(* IEC 61131-3 sources: motion-safety-bench/plc, 16 files *)

(* ---- Enumerations.st ---- *)
TYPE E_MachineMode :
(
    MODE_OFF        := 0,
    MODE_INIT       := 1,
    MODE_HOMING     := 2,
    MODE_MANUAL_JOG := 3,
    MODE_AUTO       := 4,
    MODE_FAULT      := 5,
    MODE_RESET      := 6
);
END_TYPE

TYPE E_AxisState :
(
    AXIS_DISABLED           := 0,
    AXIS_STANDSTILL         := 1,
    AXIS_HOMING             := 2,
    AXIS_DISCRETE_MOTION    := 3,
    AXIS_CONTINUOUS_MOTION  := 4,
    AXIS_STOPPING           := 5,
    AXIS_ERRORSTOP          := 6
);
END_TYPE

TYPE E_AlarmSeverity :
(
    SEV_INFO        := 0,
    SEV_WARNING     := 1,
    SEV_FAULT       := 2,
    SEV_CRITICAL    := 3
);
END_TYPE

TYPE E_AlarmState :
(
    ALARM_INACTIVE      := 0,
    ALARM_ACTIVE        := 1,
    ALARM_ACKNOWLEDGED  := 2,
    ALARM_CLEARED       := 3
);
END_TYPE

TYPE E_CommandType :
(
    CMD_NONE                := 0,
    CMD_MODE_REQUEST        := 1,
    CMD_JOG_POSITIVE        := 2,
    CMD_JOG_NEGATIVE        := 3,
    CMD_MOVE_ABSOLUTE       := 4,
    CMD_MOVE_RELATIVE       := 5,
    CMD_STOP                := 6,
    CMD_RESET               := 7,
    CMD_HOME                := 8,
    CMD_ACK_ALARM           := 9,
    CMD_RESET_ALL_ALARMS    := 10
);
END_TYPE

TYPE E_CommandStatus :
(
    CMDSTAT_IDLE        := 0,
    CMDSTAT_PENDING     := 1,
    CMDSTAT_EXECUTING   := 2,
    CMDSTAT_DONE        := 3,
    CMDSTAT_ERROR       := 4
);
END_TYPE

TYPE E_HomingState :
(
    HOM_IDLE            := 0,
    HOM_SEEKING_SWITCH  := 1,
    HOM_BACKING_OFF     := 2,
    HOM_SEEKING_INDEX   := 3,
    HOM_SETTING_POS     := 4,
    HOM_COMPLETE        := 5,
    HOM_ERROR           := 6
);
END_TYPE

TYPE E_TraceSource :
(
    TRACE_MODE      := 0,
    TRACE_AXIS      := 1,
    TRACE_HOMING    := 2,
    TRACE_SAFETY    := 3,
    TRACE_ALARM     := 4,
    TRACE_COMMAND   := 5,
    TRACE_CONFIG    := 6,
    TRACE_TEST      := 7
);
END_TYPE

TYPE E_TestPhase :
(
    TEST_IDLE       := 0,
    TEST_SETUP      := 1,
    TEST_EXECUTE    := 2,
    TEST_SETTLE     := 3,
    TEST_VERIFY     := 4,
    TEST_TEARDOWN   := 5,
    TEST_DONE       := 6
);
END_TYPE

TYPE E_TestResult :
(
    TRES_NOT_RUN    := 0,
    TRES_RUNNING    := 1,
    TRES_PASS       := 2,
    TRES_FAIL       := 3,
    TRES_TIMEOUT    := 4
);
END_TYPE

(* ---- Structures.st ---- *)
TYPE ST_AxisConfig :
STRUCT
    fMaxVelocity : LREAL := 500.0;
    fMaxAcceleration : LREAL := 2000.0;
    fMaxDeceleration : LREAL := 2000.0;
    fJerkLimit : LREAL := 10000.0;
    fSoftLimitPositive : LREAL := 300.0;
    fSoftLimitNegative : LREAL := -10.0;
    fHomingVelocity : LREAL := 50.0;
    fHomingBackoffVelocity : LREAL := 10.0;
    bHomingDirectionPositive : BOOL := FALSE;
    fHomeOffset : LREAL := 0.0;
    fPositionErrorLimit : LREAL := 2.0;
    fJogVelocity : LREAL := 100.0;
END_STRUCT
END_TYPE

TYPE ST_AxisStatus :
STRUCT
    fActualPosition : LREAL;
    fActualVelocity : LREAL;
    fActualTorque : LREAL;
    eAxisState : E_AxisState;
    bEnabled : BOOL;
    bHomed : BOOL;
    bInMotion : BOOL;
    bError : BOOL;
    nErrorCode : UDINT;
    bPositiveLimitActive : BOOL;
    bNegativeLimitActive : BOOL;
END_STRUCT
END_TYPE

TYPE ST_SafetyConfig :
STRUCT
    tEStopDebounceTime : TIME := T#100MS;
    tRelayDiscrepancyWindow : TIME := T#500MS;
    tLimitDebounceTime : TIME := T#50MS;
    tStuckSensorTimeout : TIME := T#5S;
END_STRUCT
END_TYPE

TYPE ST_SafetyStatus :
STRUCT
    bSafeToRun : BOOL;
    bEStopActive : BOOL;
    bSafetyRelayOK : BOOL;
    bRelayDiscrepancy : BOOL;
    bAnyLimitTripped : BOOL;
    abLimitPosActive : ARRAY[1..2] OF BOOL;
    abLimitNegActive : ARRAY[1..2] OF BOOL;
    nSafetyStatusWord : UINT;
END_STRUCT
END_TYPE

TYPE ST_Alarm :
STRUCT
    nID : UINT;
    eSeverity : E_AlarmSeverity;
    eState : E_AlarmState;
    sMessage : STRING(80);
    sSource : STRING(40);
    tRaiseTime : DT;
    tAckTime : DT;
    tClearTime : DT;
    bRequiresAck : BOOL;
    bSelfClearing : BOOL;
END_STRUCT
END_TYPE

TYPE ST_HMICommand :
STRUCT
    eCommandType : E_CommandType;
    nAxisIndex : UINT;
    fValue1 : LREAL;
    fValue2 : LREAL;
    eTargetMode : E_MachineMode;
    nAlarmID : UINT;
    bExecute : BOOL;
END_STRUCT
END_TYPE

TYPE ST_MotionCommand :
STRUCT
    eType : E_CommandType;
    nAxisIndex : UINT;
    fTargetPosition : LREAL;
    fDistance : LREAL;
    fVelocity : LREAL;
    bJogPositive : BOOL;
    bJogNegative : BOOL;
    bExecute : BOOL;
    eStatus : E_CommandStatus;
END_STRUCT
END_TYPE

TYPE ST_TraceEvent :
STRUCT
    tTimestamp : DT;
    eSource : E_TraceSource;
    nEventID : UINT;
    sDescription : STRING(120);
    fValue : LREAL;
END_STRUCT
END_TYPE

TYPE ST_ModePermits :
STRUCT
    bAllowMotion : BOOL;
    bAllowJog : BOOL;
    bAllowHoming : BOOL;
    bAllowAutoStart : BOOL;
    bAllowModeChange : BOOL;
    bAllowConfigEdit : BOOL;
    bAllowAlarmReset : BOOL;
END_STRUCT
END_TYPE

TYPE ST_TimingConfig :
STRUCT
    tInitTimeout : TIME := T#10S;
    tHomingTimeout : TIME := T#60S;
    tHomingStepTimeout : TIME := T#15S;
    nHomingMaxRetries : UINT := 2;
    tCommandTimeout : TIME := T#5S;
    tTestSettleTime : TIME := T#500MS;
    tTestStepTimeout : TIME := T#30S;
END_STRUCT
END_TYPE

TYPE ST_TraceConfig :
STRUCT
    nBufferSize : UINT := 1000;
    nDisplayCount : UINT := 20;
    nPendingQueueMax : UINT := 50;
END_STRUCT
END_TYPE

TYPE ST_AlarmConfig :
STRUCT
    nMaxActiveAlarms : UINT := 32;
    nMaxAlarmHistory : UINT := 200;
END_STRUCT
END_TYPE

TYPE ST_MachineConfig :
STRUCT
    bSimulationMode : BOOL := TRUE;
    astAxisConfig : ARRAY[1..2] OF ST_AxisConfig;
    stSafetyConfig : ST_SafetyConfig;
    stTimingConfig : ST_TimingConfig;
    stTraceConfig : ST_TraceConfig;
    stAlarmConfig : ST_AlarmConfig;
    nAxisCount : UINT := 2;
END_STRUCT
END_TYPE

TYPE ST_TestResult :
STRUCT
    nTestID : UINT;
    sTestName : STRING(80);
    eResult : E_TestResult;
    sExpected : STRING(120);
    sActual : STRING(120);
    tDuration : TIME;
    tTimestamp : DT;
END_STRUCT
END_TYPE

TYPE ST_HMIData :
STRUCT
    eCurrentMode : E_MachineMode;
    stModePermits : ST_ModePermits;
    astAxisStatus : ARRAY[1..2] OF ST_AxisStatus;
    stSafetyStatus : ST_SafetyStatus;
    astActiveAlarms : ARRAY[1..32] OF ST_Alarm;
    nActiveAlarmCount : UINT;
    eHighestSeverity : E_AlarmSeverity;
    astRecentEvents : ARRAY[1..20] OF ST_TraceEvent;
    eHomingState : E_HomingState;
    bSimulationMode : BOOL;
    bHMIDataStale : BOOL;
    nCycleCount : UDINT;
END_STRUCT
END_TYPE

TYPE ST_VirtualIO :
STRUCT
    bEStop : BOOL := TRUE;
    bSafetyRelayFB : BOOL := TRUE;
    abHomeSwitch : ARRAY[1..2] OF BOOL;
    abLimitPos : ARRAY[1..2] OF BOOL := [TRUE, TRUE];
    abLimitNeg : ARRAY[1..2] OF BOOL := [TRUE, TRUE];
    bSensor1 : BOOL;
    bSensor2 : BOOL;
    bReadyLamp : BOOL;
    bFaultLamp : BOOL;
    bMotionLamp : BOOL;
    bHomedLamp : BOOL;
    bSafetyRelayCmd : BOOL;
END_STRUCT
END_TYPE

(* ---- GVL_Constants.st ---- *)
VAR_GLOBAL CONSTANT
    cMAX_AXES : UINT := 2;
    cMAX_ALARMS : UINT := 32;
    cMAX_ALARM_HISTORY : UINT := 200;
    cTRACE_BUFFER_SIZE : UINT := 1000;
    cTRACE_DISPLAY_COUNT : UINT := 20;
    cTRACE_PENDING_MAX : UINT := 50;
    cMAX_TESTS : UINT := 50;
END_VAR

(* ---- GVL_IO.st ---- *)
(*
    This is the ONLY file with AT% addresses.
    All other files use symbolic names.
*)
VAR_GLOBAL
    (* Inputs *)
    bPhysEStop           AT %IX0.0 : BOOL;
    bPhysSafetyRelayFB   AT %IX0.1 : BOOL;
    bPhysHomeSwitch1     AT %IX0.2 : BOOL;
    bPhysHomeSwitch2     AT %IX0.3 : BOOL;
    bPhysLimitPos1       AT %IX0.4 : BOOL;
    bPhysLimitNeg1       AT %IX0.5 : BOOL;
    bPhysLimitPos2       AT %IX0.6 : BOOL;
    bPhysLimitNeg2       AT %IX0.7 : BOOL;
    bPhysGuardDoorClosed AT %IX1.0 : BOOL;
    bPhysSTOHealthy      AT %IX1.1 : BOOL;
    bPhysDriveReady1     AT %IX1.2 : BOOL;
    bPhysDriveReady2     AT %IX1.3 : BOOL;
    bPhysDriveFault1     AT %IX1.4 : BOOL;
    bPhysDriveFault2     AT %IX1.5 : BOOL;
    bPhysEncoderHealthy1 AT %IX1.6 : BOOL;
    bPhysEncoderHealthy2 AT %IX1.7 : BOOL;
    bPhysEtherCATOK      AT %IX2.0 : BOOL;
    bPhysWatchdogOK      AT %IX2.1 : BOOL;

    (* Outputs *)
    bPhysReadyLamp       AT %QX0.0 : BOOL;
    bPhysFaultLamp       AT %QX0.1 : BOOL;
    bPhysMotionLamp      AT %QX0.2 : BOOL;
    bPhysHomedLamp       AT %QX0.3 : BOOL;
    bPhysSafetyRelayCmd  AT %QX0.4 : BOOL;
END_VAR

(* ---- GVL_VirtualIO.st ---- *)
VAR_GLOBAL
    (* Written by TestHarness or simulation environment. bSimulationMode must be TRUE. *)
    stVirtualIO : ST_VirtualIO;
END_VAR

(* ---- AlarmManager.st ---- *)
FUNCTION_BLOCK FB_AlarmManager
VAR_INPUT
    stSafetyStatus      : ST_SafetyStatus;
    bAnyAxisError       : BOOL;
    bHomingError        : BOOL;
    bConfigInvalid      : BOOL;
    bAckRequested       : BOOL;
    nAckAlarmID         : UINT;
    bResetAllRequested  : BOOL;
END_VAR

VAR_OUTPUT
    bAnyFaultActive     : BOOL;
    bAnyAlarmActive     : BOOL;
    nActiveAlarmCount   : UINT;
    eHighestSeverity    : E_AlarmSeverity;
    astActiveAlarms     : ARRAY[1..32] OF ST_Alarm;
END_VAR

VAR
    astAlarmBuffer      : ARRAY[1..32] OF ST_Alarm;
    astHistory          : ARRAY[1..200] OF ST_Alarm;
    nWriteIdx           : UINT;
    nHistoryIdx         : UINT;
END_VAR

(* ========== CONDITION EVALUATION ========== *)
METHOD EvaluateConditions
(* Method: EvaluateConditions — Purpose: Check all alarm source conditions, raise alarms as needed *)
(* TODO: IF NOT stSafetyStatus.bSafeToRun AND stSafetyStatus.bEStopActive THEN RaiseAlarm(1001, SEV_CRITICAL, 'E-stop active', 'SafetyManager', TRUE) *)
(* TODO: IF stSafetyStatus.bRelayDiscrepancy THEN RaiseAlarm(1002, SEV_CRITICAL, 'Safety relay discrepancy', 'SafetyManager', TRUE) *)
(* TODO: IF stSafetyStatus.bAnyLimitTripped THEN RaiseAlarm(1003, SEV_FAULT, 'Limit switch tripped', 'SafetyManager', TRUE) *)
(* TODO: IF bAnyAxisError THEN RaiseAlarm(2001, SEV_FAULT, 'Axis error', 'AxisManager', TRUE) *)
(* TODO: IF bHomingError THEN RaiseAlarm(3001, SEV_FAULT, 'Homing failed', 'HomingManager', TRUE) *)
END_METHOD

(* ========== OUTPUTS ========== *)
METHOD UpdateOutputs
(* Method: UpdateOutputs — Purpose: Update bAnyFaultActive, counts, highest severity *)
(* TODO: iterate astAlarmBuffer, count ACTIVE alarms, find highest severity *)
(* TODO: set bAnyFaultActive := any alarm with eSeverity >= SEV_FAULT is ACTIVE and unacknowledged *)
(* TODO: copy active alarms to astActiveAlarms output *)
END_METHOD

(* ========== RAISE ALARM ========== *)
METHOD RaiseAlarm
VAR_INPUT
    nID         : UINT;
    eSeverity   : E_AlarmSeverity;
    sMessage    : STRING(80);
    sSource     : STRING(40);
    bRequiresAck: BOOL;
END_VAR
(* Method: RaiseAlarm — Purpose: Add or update alarm in buffer with timestamp *)
(* TODO: check if alarm nID already active, if not find empty slot and populate *)
(* TODO: set tRaiseTime := NOW_DT(), eState := ALARM_ACTIVE *)
END_METHOD

(* ========== ACKNOWLEDGE ALARM ========== *)
METHOD AcknowledgeAlarm
VAR_INPUT
    nAlarmID : UINT;
END_VAR
(* Method: AcknowledgeAlarm — Purpose: Transition alarm from ACTIVE to ACKNOWLEDGED *)
(* TODO: find alarm by nID, if eState=ALARM_ACTIVE set eState:=ALARM_ACKNOWLEDGED, tAckTime:=NOW_DT() *)
END_METHOD

(* ========== RESET ALARM ========== *)
METHOD ResetAlarm
VAR_INPUT
    nAlarmID : UINT;
END_VAR
(* Method: ResetAlarm — Purpose: Clear alarm if condition is gone *)
(* TODO: find alarm by nID, if NOT bRequiresAck or already ACKNOWLEDGED, set eState:=ALARM_CLEARED *)
END_METHOD

(* ========== RESET ALL ALARMS ========== *)
METHOD ResetAllAlarms
(* Method: ResetAllAlarms — Purpose: Clear all clearable alarms *)
(* TODO: iterate buffer, call ResetAlarm on each *)
END_METHOD

END_FUNCTION_BLOCK

(* ---- CommandParser.st ---- *)
FUNCTION_BLOCK FB_CommandParser
VAR_INPUT
    stHMICommand    : ST_HMICommand;
    eCurrentMode    : E_MachineMode;
    stModePermits   : ST_ModePermits;
    stSafetyStatus  : ST_SafetyStatus;
END_VAR

VAR_OUTPUT
    eRequestedMode      : E_MachineMode;
    stMotionCommand     : ST_MotionCommand;
    bStartHoming        : BOOL;
    bAbortHoming        : BOOL;
    bAckRequested       : BOOL;
    nAckAlarmID         : UINT;
    bResetRequested     : BOOL;
    bResetAllRequested  : BOOL;
    eLastCommandStatus  : E_CommandStatus;
    sLastCommandError   : STRING(120);
END_VAR

VAR
    eProcessingState    : E_CommandStatus;
    rtrigExecute        : R_TRIG;
    nCommandCounter     : UDINT;
    nRejectedCounter    : UDINT;
END_VAR

METHOD Cyclic
(* Method: Cyclic - Purpose: Detect rising edge on bExecute, validate, route command *)

rtrigExecute(CLK := stHMICommand.bExecute);

IF rtrigExecute.Q THEN
    nCommandCounter := nCommandCounter + 1;
    IF ValidateCommand() THEN
        eLastCommandStatus := CMDSTAT_EXECUTING;
        sLastCommandError := '';

        CASE stHMICommand.eCommandType OF
            CMD_MODE_REQUEST:
                eRequestedMode := stHMICommand.eTargetMode;

            CMD_JOG_POSITIVE, CMD_JOG_NEGATIVE, CMD_MOVE_ABSOLUTE, CMD_MOVE_RELATIVE, CMD_STOP:
                stMotionCommand.eType := stHMICommand.eCommandType;
                stMotionCommand.nAxisIndex := stHMICommand.nAxisIndex;
                stMotionCommand.fTargetPosition := stHMICommand.fValue1;
                stMotionCommand.fDistance := stHMICommand.fValue1;
                stMotionCommand.fVelocity := stHMICommand.fValue2;
                stMotionCommand.bExecute := TRUE;

            CMD_HOME:
                bStartHoming := TRUE;

            CMD_RESET:
                bResetRequested := TRUE;

            CMD_ACK_ALARM:
                bAckRequested := TRUE;
                nAckAlarmID := stHMICommand.nAlarmID;

            CMD_RESET_ALL_ALARMS:
                bResetAllRequested := TRUE;
        END_CASE
    ELSE
        eLastCommandStatus := CMDSTAT_ERROR;
        nRejectedCounter := nRejectedCounter + 1;
    END_IF
ELSE
    (* Reset single-cycle triggers *)
    bStartHoming := FALSE;
    bResetRequested := FALSE;
    bAckRequested := FALSE;
    bResetAllRequested := FALSE;
    IF stMotionCommand.eType <> CMD_JOG_POSITIVE AND stMotionCommand.eType <> CMD_JOG_NEGATIVE THEN
        stMotionCommand.bExecute := FALSE;
    ELSE
        (* Keep jog active if bExecute is still true in the input struct *)
        stMotionCommand.bExecute := stHMICommand.bExecute;
    END_IF
END_IF

END_METHOD

METHOD ValidateCommand : BOOL
(* Method: ValidateCommand - Purpose: Check if command allowed in current mode and safety state *)

ValidateCommand := FALSE;

CASE stHMICommand.eCommandType OF
    CMD_MODE_REQUEST:
        IF stModePermits.bAllowModeChange THEN
            ValidateCommand := TRUE;
        ELSE
            sLastCommandError := 'Mode change not permitted';
        END_IF

    CMD_JOG_POSITIVE, CMD_JOG_NEGATIVE:
        IF stModePermits.bAllowJog AND stSafetyStatus.bSafeToRun THEN
            ValidateCommand := TRUE;
        ELSE
            sLastCommandError := 'Jog not permitted or safety not OK';
        END_IF

    CMD_MOVE_ABSOLUTE, CMD_MOVE_RELATIVE:
        IF stModePermits.bAllowMotion AND stSafetyStatus.bSafeToRun THEN
            ValidateCommand := TRUE;
        ELSE
            sLastCommandError := 'Motion not permitted or safety not OK';
        END_IF

    CMD_STOP:
        ValidateCommand := TRUE;

    CMD_HOME:
        IF stModePermits.bAllowHoming THEN
            ValidateCommand := TRUE;
        ELSE
            sLastCommandError := 'Homing not permitted';
        END_IF

    CMD_RESET, CMD_ACK_ALARM, CMD_RESET_ALL_ALARMS:
        IF stModePermits.bAllowAlarmReset THEN
            ValidateCommand := TRUE;
        ELSE
             sLastCommandError := 'Reset not permitted';
        END_IF

    CMD_NONE:
        ValidateCommand := TRUE;
END_CASE

END_METHOD

END_FUNCTION_BLOCK

(* ---- ConfigPackage.st ---- *)
FUNCTION_BLOCK FB_ConfigPackage
VAR_OUTPUT
    stMachineConfig : ST_MachineConfig;
    bSimulationMode : BOOL;
    bConfigValid    : BOOL;
    bConfigChanged  : BOOL;
END_VAR

VAR
    bInitialized    : BOOL;
    stPrevConfig    : ST_MachineConfig;
END_VAR

(* ========== CYCLIC PROCESSING ========== *)
METHOD Cyclic
(* Method: Cyclic — Purpose: Detect config changes, validate on change, set bConfigValid *)
(* TODO: compare stMachineConfig to stPrevConfig, if different set bConfigChanged, call ValidateAll *)
(* TODO: set bSimulationMode := stMachineConfig.bSimulationMode *)
END_METHOD

(* ========== DEFAULT CONFIGURATION ========== *)
METHOD LoadDefaults
(* Method: LoadDefaults — Purpose: Set all stMachineConfig fields to SDS default values *)
(* TODO: set stMachineConfig.bSimulationMode := TRUE *)
(* TODO: set stMachineConfig.nAxisCount := 2 *)
(* TODO: set axis config defaults per ST_AxisConfig field defaults from SDS *)
(* TODO: set stMachineConfig.stSafetyConfig to ST_SafetyConfig defaults *)
(* TODO: set stMachineConfig.stTimingConfig to ST_TimingConfig defaults *)
(* TODO: set bInitialized := TRUE *)
END_METHOD

(* ========== VALIDATION ========== *)
METHOD ValidateAll : BOOL
(* Method: ValidateAll — Purpose: Check all parameters, clamp or flag invalid values *)
(* Returns TRUE if all valid *)
(* TODO: check fMaxVelocity > 0 for each axis *)
(* TODO: check fSoftLimitPositive > fSoftLimitNegative for each axis *)
(* TODO: check all TIME values > T#0S *)
(* TODO: set bConfigValid := result *)
END_METHOD

(* ========== ACCESSORS ========== *)
METHOD GetAxisConfig : ST_AxisConfig
VAR_INPUT
    nAxisIndex : UINT;
END_VAR
(* Method: GetAxisConfig — Purpose: Return config for specific axis index *)
(* TODO: bounds check nAxisIndex against cMAX_AXES, return stMachineConfig.astAxisConfig[nAxisIndex] *)
END_METHOD

END_FUNCTION_BLOCK

(* ---- HMIModel.st ---- *)
FUNCTION_BLOCK FB_HMIModel
VAR_INPUT
    eCurrentMode : E_MachineMode;
    stModePermits : ST_ModePermits;
    astAxisStatus : ARRAY[1..2] OF ST_AxisStatus;
    stSafetyStatus : ST_SafetyStatus;
    astActiveAlarms : ARRAY[1..32] OF ST_Alarm;
    nActiveAlarmCount : UINT;
    eHighestSeverity : E_AlarmSeverity;
    astRecentEvents : ARRAY[1..20] OF ST_TraceEvent;
    eHomingState : E_HomingState;
    bSimulationMode : BOOL;
    bPLCHeartbeat : BOOL;
END_VAR
VAR_OUTPUT
    stHMIData : ST_HMIData;
    stHMICommand : ST_HMICommand;
END_VAR
VAR
    tonDataStale : TON;
    bPreviousHeartbeat : BOOL;
    bHeartbeatChanged : BOOL;
END_VAR

bHeartbeatChanged := bPLCHeartbeat <> bPreviousHeartbeat;
IF bHeartbeatChanged THEN
    bPreviousHeartbeat := bPLCHeartbeat;
END_IF
tonDataStale(IN := NOT bHeartbeatChanged, PT := T#2S);

stHMIData.eCurrentMode := eCurrentMode;
stHMIData.stModePermits := stModePermits;
stHMIData.astAxisStatus := astAxisStatus;
stHMIData.stSafetyStatus := stSafetyStatus;
stHMIData.astActiveAlarms := astActiveAlarms;
stHMIData.nActiveAlarmCount := nActiveAlarmCount;
stHMIData.eHighestSeverity := eHighestSeverity;
stHMIData.astRecentEvents := astRecentEvents;
stHMIData.eHomingState := eHomingState;
stHMIData.bSimulationMode := bSimulationMode;
stHMIData.bHMIDataStale := tonDataStale.Q;
stHMIData.nCycleCount := stHMIData.nCycleCount + 1;

END_FUNCTION_BLOCK

(* ---- ModeManager.st ---- *)
FUNCTION_BLOCK FB_ModeManager
VAR_INPUT
    stSafetyStatus      : ST_SafetyStatus;
    bAnyFaultActive     : BOOL;
    bAllAxesReady       : BOOL;
    bAllAxesHomed       : BOOL;
    eRequestedMode      : E_MachineMode;
    bResetRequested     : BOOL;
END_VAR

VAR_OUTPUT
    eCurrentMode            : E_MachineMode;
    ePreviousMode           : E_MachineMode;
    bModeTransitionActive   : BOOL;
    stModePermits           : ST_ModePermits;
END_VAR

VAR
    eInternalMode       : E_MachineMode;
    tonInitTimeout      : TON;
    tonHomingTimeout    : TON;
    bTransitionValid    : BOOL;
    rtrigModeRequest    : R_TRIG;
    rtrigResetRequest   : R_TRIG;
END_VAR

(* ========== CYCLIC PROCESSING ========== *)
METHOD Cyclic
(* Method: Cyclic — Purpose: Evaluate state machine, apply safety override, update permits *)

(* ========== SAFETY OVERRIDE (runs before CASE) ========== *)
(* TODO: IF NOT stSafetyStatus.bSafeToRun AND eInternalMode <> MODE_OFF AND eInternalMode <> MODE_FAULT THEN *)
(*           ePreviousMode := eInternalMode; eInternalMode := MODE_FAULT; END_IF *)

(* ========== STATE MACHINE ========== *)
CASE eInternalMode OF
    MODE_OFF:
        (* TODO: if StartCommand received and power healthy, transition to MODE_INIT *)
    MODE_INIT:
        (* TODO: run init timeout timer *)
        (* TODO: if init complete (axes ready, config valid, safety OK, no faults): stay in INIT awaiting homing request *)
        (* TODO: if HomingRequest and no faults: transition to MODE_HOMING *)
        (* TODO: if timeout: transition to MODE_FAULT *)
    MODE_HOMING:
        (* TODO: run homing timeout timer *)
        (* TODO: if bAllAxesHomed: transition to MODE_MANUAL_JOG *)
        (* TODO: if timeout or fault: transition to MODE_FAULT *)
    MODE_MANUAL_JOG:
        (* TODO: if AutoRequest and bAllAxesHomed: transition to MODE_AUTO *)
        (* TODO: if ReHomeRequest: transition to MODE_HOMING *)
        (* TODO: if bAnyFaultActive: transition to MODE_FAULT *)
    MODE_AUTO:
        (* TODO: if ManualRequest: transition to MODE_MANUAL_JOG (after axis stops) *)
        (* TODO: if bAnyFaultActive: transition to MODE_FAULT *)
    MODE_FAULT:
        (* TODO: latch — only exit via RESET when operator acknowledges *)
    MODE_RESET:
        (* TODO: 2s settle, re-check, transition to MODE_INIT or back to MODE_FAULT *)
END_CASE

(* TODO: eCurrentMode := eInternalMode *)
(* TODO: call UpdatePermits *)
END_METHOD

(* ========== TRANSITION VALIDATION ========== *)
METHOD ValidateTransition : BOOL
VAR_INPUT
    eFrom : E_MachineMode;
    eTo   : E_MachineMode;
END_VAR
(* Method: ValidateTransition — Purpose: Return TRUE if transition is valid per state table *)
(* TODO: CASE eFrom with nested IF on eTo checking all valid transitions from SDS Section 4.1 *)
END_METHOD

(* ========== MODE PERMITS ========== *)
METHOD UpdatePermits
(* Method: UpdatePermits — Purpose: Set stModePermits fields based on eCurrentMode *)
(* TODO: CASE eCurrentMode:
    MODE_MANUAL_JOG: bAllowMotion:=TRUE, bAllowJog:=TRUE, bAllowHoming:=TRUE, bAllowAutoStart:=TRUE
    MODE_AUTO: bAllowMotion:=TRUE, bAllowAutoStart:=FALSE (running), bAllowJog:=FALSE
    MODE_OFF: bAllowConfigEdit:=TRUE, rest FALSE
    all others: all FALSE except bAllowAlarmReset in FAULT *)
END_METHOD

END_FUNCTION_BLOCK

(* ---- SafetyManager.st ---- *)
FUNCTION_BLOCK FB_SafetyManager
VAR_INPUT
    bSimulationMode     : BOOL;
    stConfig            : ST_SafetyConfig;
    abDriveReady        : ARRAY[1..2] OF BOOL;
END_VAR

VAR_OUTPUT
    stSafetyStatus      : ST_SafetyStatus;
    bSafeToRun          : BOOL;
    bEStopActive        : BOOL;
    bAnyLimitTripped    : BOOL;
END_VAR

VAR
    bEStopRaw           : BOOL;
    bRelayFBRaw         : BOOL;
    abLimitPosRaw       : ARRAY[1..2] OF BOOL;
    abLimitNegRaw       : ARRAY[1..2] OF BOOL;
    tonEStopDebounce    : TON;
    tonRelayDiscrep     : TON;
    bRelayDiscrepancy   : BOOL;
END_VAR

(* ========== CYCLIC PROCESSING ========== *)
METHOD Cyclic
(* Method: Cyclic — Purpose: Read inputs, apply debounce, compute bSafeToRun *)
(* Step 1: call ReadInputs to populate raw signals *)
(* Step 2: apply debounce timers *)
(* Step 3: check relay discrepancy *)
(* TODO: bSafeToRun := bEStopRaw AND bRelayFBRaw AND NOT bRelayDiscrepancy AND NOT bAnyLimitTripped *)
(* TODO: populate stSafetyStatus fields *)
(* TODO: set nSafetyStatusWord as bitfield of key signals *)
END_METHOD

(* ========== INPUT SELECTION ========== *)
METHOD ReadInputs
(* Method: ReadInputs — Purpose: Select virtual or physical I/O based on bSimulationMode *)
(* TODO: IF bSimulationMode THEN read from GVL_VirtualIO.stVirtualIO ELSE read from GVL_IO *)
(* Note: E-stop and limits are NC logic — TRUE = healthy, FALSE = activated *)
END_METHOD

END_FUNCTION_BLOCK

(* ---- TestHarness.st ---- *)
FUNCTION_BLOCK FB_TestHarness
VAR_INPUT
    bRunTest : BOOL;
    nTestID : UINT;
    bRunAllTests : BOOL;
    eCurrentMode : E_MachineMode;
    astAxisStatus : ARRAY[1..2] OF ST_AxisStatus;
    stSafetyStatus : ST_SafetyStatus;
    nActiveAlarmCount : UINT;
    nTraceEventCount : UDINT;
    bSimulationMode : BOOL;
END_VAR
VAR_OUTPUT
    stHMICommand : ST_HMICommand;
    stTestResult : ST_TestResult;
    astTestSummary : ARRAY[1..50] OF ST_TestResult;
    nTestsRun : UINT;
    nTestsPassed : UINT;
    nTestsFailed : UINT;
    nCurrentTestID : UINT;
    bTestSuiteRunning : BOOL;
    bTestSuiteComplete : BOOL;
END_VAR
VAR
    eTestPhase : E_TestPhase;
    nTestStep : UINT;
    nCyclesInPhase : UDINT;
    rtrigRunTest : R_TRIG;
    rtrigRunAll : R_TRIG;
    bRunSuite : BOOL;
    bVerificationPassed : BOOL;
    bFaultObserved : BOOL;
    fInitialPosition : LREAL;
    fExpectedPosition : LREAL;
    fPeakPosition : LREAL;
    fLowPosition : LREAL;
    sTestName : STRING(80);
    sExpected : STRING(120);
    sActual : STRING(120);
END_VAR

rtrigRunTest(CLK := bRunTest);
rtrigRunAll(CLK := bRunAllTests);

(* All command edges are one scan wide unless explicitly held for jog. *)
stHMICommand.bExecute := FALSE;

IF NOT bSimulationMode THEN
    bTestSuiteRunning := FALSE;
    eTestPhase := TEST_IDLE;
ELSE
    IF rtrigRunAll.Q THEN
        nTestsRun := 0;
        nTestsPassed := 0;
        nTestsFailed := 0;
        nCurrentTestID := 1;
        bRunSuite := TRUE;
        bTestSuiteRunning := TRUE;
        bTestSuiteComplete := FALSE;
        eTestPhase := TEST_SETUP;
        nTestStep := 0;
        nCyclesInPhase := 0;
    ELSIF rtrigRunTest.Q AND (nTestID >= 1) AND (nTestID <= 16) THEN
        nCurrentTestID := nTestID;
        bRunSuite := FALSE;
        bTestSuiteRunning := TRUE;
        bTestSuiteComplete := FALSE;
        eTestPhase := TEST_SETUP;
        nTestStep := 0;
        nCyclesInPhase := 0;
    END_IF

    IF bTestSuiteRunning THEN
        nCyclesInPhase := nCyclesInPhase + 1;

        CASE eTestPhase OF
            TEST_SETUP:
                GVL_VirtualIO.stVirtualIO.bEStop := TRUE;
                GVL_VirtualIO.stVirtualIO.bSafetyRelayFB := TRUE;
                GVL_VirtualIO.stVirtualIO.bGuardDoorClosed := TRUE;
                GVL_VirtualIO.stVirtualIO.bSTOHealthy := TRUE;
                GVL_VirtualIO.stVirtualIO.bEtherCATOK := TRUE;
                GVL_VirtualIO.stVirtualIO.bWatchdogOK := TRUE;
                GVL_VirtualIO.stVirtualIO.abLimitPos[1] := TRUE;
                GVL_VirtualIO.stVirtualIO.abLimitNeg[1] := TRUE;
                GVL_VirtualIO.stVirtualIO.abLimitPos[2] := TRUE;
                GVL_VirtualIO.stVirtualIO.abLimitNeg[2] := TRUE;
                GVL_VirtualIO.stVirtualIO.abDriveReady[1] := TRUE;
                GVL_VirtualIO.stVirtualIO.abDriveReady[2] := TRUE;
                GVL_VirtualIO.stVirtualIO.abDriveFault[1] := FALSE;
                GVL_VirtualIO.stVirtualIO.abDriveFault[2] := FALSE;
                GVL_VirtualIO.stVirtualIO.abEncoderHealthy[1] := TRUE;
                GVL_VirtualIO.stVirtualIO.abEncoderHealthy[2] := TRUE;
                GVL_VirtualIO.stVirtualIO.abFollowingError[1] := FALSE;
                GVL_VirtualIO.stVirtualIO.abFollowingError[2] := FALSE;
                GVL_VirtualIO.stVirtualIO.abHomeSwitch[1] := FALSE;
                GVL_VirtualIO.stVirtualIO.abHomeSwitch[2] := FALSE;

                fInitialPosition := astAxisStatus[1].fActualPosition;
                fExpectedPosition := fInitialPosition;
                fPeakPosition := fInitialPosition;
                fLowPosition := fInitialPosition;
                bVerificationPassed := FALSE;
                bFaultObserved := FALSE;

                CASE nCurrentTestID OF
                    1:
                        sTestName := 'TR01 Startup and Homing';
                        sExpected := 'Safe startup reaches MANUAL with both axes homed';
                    2:
                        sTestName := 'TR02 Absolute Move';
                        sExpected := 'Axis 1 reaches 100.0 mm';
                    3:
                        sTestName := 'TR03 Relative Move';
                        sExpected := 'Axis 1 advances by 50.0 mm';
                        fExpectedPosition := fInitialPosition + 50.0;
                    4:
                        sTestName := 'TR04 Jog Positive and Negative';
                        sExpected := 'Axis jogs both directions and stops on release';
                    5:
                        sTestName := 'TR05 Positive Limit Switch';
                        sExpected := 'Positive limit stops motion, enters FAULT, recovers';
                    6:
                        sTestName := 'TR06 Negative Limit Switch';
                        sExpected := 'Negative limit stops motion, enters FAULT, recovers';
                    7:
                        sTestName := 'TR07 E-stop During Motion';
                        sExpected := 'E-stop stops motion, enters FAULT, recovers';
                    8:
                        sTestName := 'TR08 Guard Door During Motion';
                        sExpected := 'Guard door inhibits motion, enters FAULT, recovers';
                    9:
                        sTestName := 'TR09 Drive Fault';
                        sExpected := 'Drive fault latches axis error and recovers through RESET';
                    10:
                        sTestName := 'TR10 Following Error';
                        sExpected := 'Following error is detected and recovered';
                    11:
                        sTestName := 'TR11 Encoder Feedback Loss';
                        sExpected := 'Feedback loss is detected and recovered';
                    12:
                        sTestName := 'TR12 EtherCAT Dropout';
                        sExpected := 'Network dropout inhibits motion and recovers';
                    13:
                        sTestName := 'TR13 Warm Restart';
                        sExpected := 'Stop/restart leaves no stale motion command';
                    14:
                        sTestName := 'TR14 Cold Restart Defaults';
                        sExpected := 'Virtual safe defaults are restored';
                    15:
                        sTestName := 'TR15 Watchdog Timeout';
                        sExpected := 'Watchdog loss enters FAULT and recovers';
                    16:
                        sTestName := 'TR16 Invalid Command Transition';
                        sExpected := 'Move command in OFF is rejected without motion';
                END_CASE

                stTestResult.nTestID := nCurrentTestID;
                stTestResult.sTestName := sTestName;
                stTestResult.sExpected := sExpected;
                stTestResult.eResult := TRES_RUNNING;
                eTestPhase := TEST_EXECUTE;
                nTestStep := 0;
                nCyclesInPhase := 0;

            TEST_EXECUTE:
                IF astAxisStatus[1].fActualPosition > fPeakPosition THEN
                    fPeakPosition := astAxisStatus[1].fActualPosition;
                END_IF
                IF astAxisStatus[1].fActualPosition < fLowPosition THEN
                    fLowPosition := astAxisStatus[1].fActualPosition;
                END_IF

                CASE nCurrentTestID OF
                    1:
                        IF nTestStep = 0 THEN
                            stHMICommand.eCommandType := CMD_MODE_REQUEST;
                            stHMICommand.eTargetMode := MODE_INIT;
                            stHMICommand.bExecute := TRUE;
                            nTestStep := 1;
                        ELSIF nTestStep = 1 THEN
                            nTestStep := 2;
                        ELSIF nTestStep = 2 THEN
                            stHMICommand.eCommandType := CMD_MODE_REQUEST;
                            stHMICommand.eTargetMode := MODE_HOMING;
                            stHMICommand.bExecute := TRUE;
                            nTestStep := 3;
                        ELSIF nTestStep = 3 THEN
                            nTestStep := 4;
                        ELSIF nTestStep = 4 THEN
                            stHMICommand.eCommandType := CMD_HOME;
                            stHMICommand.bExecute := TRUE;
                            nTestStep := 5;
                        ELSIF nCyclesInPhase = 20 THEN
                            GVL_VirtualIO.stVirtualIO.abHomeSwitch[1] := TRUE;
                        ELSIF nCyclesInPhase = 30 THEN
                            GVL_VirtualIO.stVirtualIO.abHomeSwitch[1] := FALSE;
                        ELSIF nCyclesInPhase = 40 THEN
                            GVL_VirtualIO.stVirtualIO.abHomeSwitch[1] := TRUE;
                        ELSIF nCyclesInPhase = 50 THEN
                            GVL_VirtualIO.stVirtualIO.abHomeSwitch[1] := FALSE;
                        ELSIF nCyclesInPhase = 60 THEN
                            GVL_VirtualIO.stVirtualIO.abHomeSwitch[2] := TRUE;
                        ELSIF nCyclesInPhase = 70 THEN
                            GVL_VirtualIO.stVirtualIO.abHomeSwitch[2] := FALSE;
                        ELSIF nCyclesInPhase = 80 THEN
                            GVL_VirtualIO.stVirtualIO.abHomeSwitch[2] := TRUE;
                        ELSIF nCyclesInPhase >= 120 THEN
                            eTestPhase := TEST_VERIFY;
                        END_IF

                    2:
                        IF nTestStep = 0 THEN
                            stHMICommand.eCommandType := CMD_MOVE_ABSOLUTE;
                            stHMICommand.nAxisIndex := 1;
                            stHMICommand.fValue1 := 100.0;
                            stHMICommand.fValue2 := 200.0;
                            stHMICommand.bExecute := TRUE;
                            nTestStep := 1;
                        ELSIF (NOT astAxisStatus[1].bInMotion) AND (nCyclesInPhase > 5) THEN
                            eTestPhase := TEST_VERIFY;
                        END_IF

                    3:
                        IF nTestStep = 0 THEN
                            stHMICommand.eCommandType := CMD_MOVE_RELATIVE;
                            stHMICommand.nAxisIndex := 1;
                            stHMICommand.fValue1 := 50.0;
                            stHMICommand.fValue2 := 200.0;
                            stHMICommand.bExecute := TRUE;
                            nTestStep := 1;
                        ELSIF (NOT astAxisStatus[1].bInMotion) AND (nCyclesInPhase > 5) THEN
                            eTestPhase := TEST_VERIFY;
                        END_IF

                    4:
                        stHMICommand.nAxisIndex := 1;
                        stHMICommand.fValue1 := 50.0;
                        IF nCyclesInPhase <= 50 THEN
                            stHMICommand.eCommandType := CMD_JOG_POSITIVE;
                            stHMICommand.bExecute := TRUE;
                        ELSIF (nCyclesInPhase >= 70) AND (nCyclesInPhase <= 120) THEN
                            stHMICommand.eCommandType := CMD_JOG_NEGATIVE;
                            stHMICommand.bExecute := TRUE;
                        ELSIF nCyclesInPhase >= 140 THEN
                            eTestPhase := TEST_VERIFY;
                        END_IF

                    5:
                        IF nTestStep = 0 THEN
                            stHMICommand.eCommandType := CMD_MOVE_ABSOLUTE;
                            stHMICommand.nAxisIndex := 1;
                            stHMICommand.fValue1 := 250.0;
                            stHMICommand.fValue2 := 100.0;
                            stHMICommand.bExecute := TRUE;
                            nTestStep := 1;
                        ELSIF (nTestStep = 1) AND (nCyclesInPhase >= 20) THEN
                            GVL_VirtualIO.stVirtualIO.abLimitPos[1] := FALSE;
                            IF (eCurrentMode = MODE_FAULT) AND (NOT astAxisStatus[1].bInMotion) THEN
                                bFaultObserved := TRUE;
                                GVL_VirtualIO.stVirtualIO.abLimitPos[1] := TRUE;
                                nTestStep := 2;
                            END_IF
                        ELSIF nTestStep = 2 THEN
                            stHMICommand.eCommandType := CMD_RESET;
                            stHMICommand.bExecute := TRUE;
                            nTestStep := 3;
                        ELSIF nTestStep = 3 THEN
                            nTestStep := 4;
                        ELSIF (nTestStep = 4) AND (nCyclesInPhase >= 90) THEN
                            stHMICommand.eCommandType := CMD_RESET_ALL_ALARMS;
                            stHMICommand.bExecute := TRUE;
                            nTestStep := 5;
                        ELSIF nTestStep = 5 THEN
                            nTestStep := 6;
                        ELSIF (nTestStep = 6) AND (nCyclesInPhase >= 140) THEN
                            stHMICommand.eCommandType := CMD_MODE_REQUEST;
                            stHMICommand.eTargetMode := MODE_MANUAL_JOG;
                            stHMICommand.bExecute := TRUE;
                            nTestStep := 7;
                        ELSIF (nTestStep = 7) AND (eCurrentMode = MODE_MANUAL_JOG) THEN
                            eTestPhase := TEST_VERIFY;
                        END_IF

                    6:
                        IF nTestStep = 0 THEN
                            stHMICommand.eCommandType := CMD_MOVE_ABSOLUTE;
                            stHMICommand.nAxisIndex := 1;
                            stHMICommand.fValue1 := -5.0;
                            stHMICommand.fValue2 := 100.0;
                            stHMICommand.bExecute := TRUE;
                            nTestStep := 1;
                        ELSIF (nTestStep = 1) AND (nCyclesInPhase >= 20) THEN
                            GVL_VirtualIO.stVirtualIO.abLimitNeg[1] := FALSE;
                            IF (eCurrentMode = MODE_FAULT) AND (NOT astAxisStatus[1].bInMotion) THEN
                                bFaultObserved := TRUE;
                                GVL_VirtualIO.stVirtualIO.abLimitNeg[1] := TRUE;
                                nTestStep := 2;
                            END_IF
                        ELSIF nTestStep = 2 THEN
                            stHMICommand.eCommandType := CMD_RESET;
                            stHMICommand.bExecute := TRUE;
                            nTestStep := 3;
                        ELSIF nTestStep = 3 THEN
                            nTestStep := 4;
                        ELSIF (nTestStep = 4) AND (nCyclesInPhase >= 90) THEN
                            stHMICommand.eCommandType := CMD_RESET_ALL_ALARMS;
                            stHMICommand.bExecute := TRUE;
                            nTestStep := 5;
                        ELSIF nTestStep = 5 THEN
                            nTestStep := 6;
                        ELSIF (nTestStep = 6) AND (nCyclesInPhase >= 140) THEN
                            stHMICommand.eCommandType := CMD_MODE_REQUEST;
                            stHMICommand.eTargetMode := MODE_MANUAL_JOG;
                            stHMICommand.bExecute := TRUE;
                            nTestStep := 7;
                        ELSIF (nTestStep = 7) AND (eCurrentMode = MODE_MANUAL_JOG) THEN
                            eTestPhase := TEST_VERIFY;
                        END_IF

                    7:
                        IF nTestStep = 0 THEN
                            stHMICommand.eCommandType := CMD_MOVE_ABSOLUTE;
                            stHMICommand.nAxisIndex := 1;
                            stHMICommand.fValue1 := 200.0;
                            stHMICommand.fValue2 := 100.0;
                            stHMICommand.bExecute := TRUE;
                            nTestStep := 1;
                        ELSIF (nTestStep = 1) AND (nCyclesInPhase >= 20) THEN
                            GVL_VirtualIO.stVirtualIO.bEStop := FALSE;
                            IF (eCurrentMode = MODE_FAULT) AND stSafetyStatus.bEStopActive THEN
                                bFaultObserved := TRUE;
                                GVL_VirtualIO.stVirtualIO.bEStop := TRUE;
                                nTestStep := 2;
                            END_IF
                        ELSIF nTestStep = 2 THEN
                            stHMICommand.eCommandType := CMD_RESET;
                            stHMICommand.bExecute := TRUE;
                            nTestStep := 3;
                        ELSIF nTestStep = 3 THEN
                            nTestStep := 4;
                        ELSIF (nTestStep = 4) AND (nCyclesInPhase >= 90) THEN
                            stHMICommand.eCommandType := CMD_RESET_ALL_ALARMS;
                            stHMICommand.bExecute := TRUE;
                            nTestStep := 5;
                        ELSIF nTestStep = 5 THEN
                            nTestStep := 6;
                        ELSIF (nTestStep = 6) AND (nCyclesInPhase >= 140) THEN
                            stHMICommand.eCommandType := CMD_MODE_REQUEST;
                            stHMICommand.eTargetMode := MODE_MANUAL_JOG;
                            stHMICommand.bExecute := TRUE;
                            nTestStep := 7;
                        ELSIF (nTestStep = 7) AND (eCurrentMode = MODE_MANUAL_JOG) THEN
                            eTestPhase := TEST_VERIFY;
                        END_IF

                    8:
                        IF nTestStep = 0 THEN
                            stHMICommand.eCommandType := CMD_MOVE_ABSOLUTE;
                            stHMICommand.nAxisIndex := 1;
                            stHMICommand.fValue1 := 180.0;
                            stHMICommand.fValue2 := 100.0;
                            stHMICommand.bExecute := TRUE;
                            nTestStep := 1;
                        ELSIF (nTestStep = 1) AND (nCyclesInPhase >= 20) THEN
                            GVL_VirtualIO.stVirtualIO.bGuardDoorClosed := FALSE;
                            IF (eCurrentMode = MODE_FAULT) AND stSafetyStatus.bGuardDoorOpen THEN
                                bFaultObserved := TRUE;
                                GVL_VirtualIO.stVirtualIO.bGuardDoorClosed := TRUE;
                                nTestStep := 2;
                            END_IF
                        ELSIF nTestStep = 2 THEN
                            stHMICommand.eCommandType := CMD_RESET;
                            stHMICommand.bExecute := TRUE;
                            nTestStep := 3;
                        ELSIF nTestStep = 3 THEN
                            nTestStep := 4;
                        ELSIF (nTestStep = 4) AND (nCyclesInPhase >= 90) THEN
                            stHMICommand.eCommandType := CMD_RESET_ALL_ALARMS;
                            stHMICommand.bExecute := TRUE;
                            nTestStep := 5;
                        ELSIF nTestStep = 5 THEN
                            nTestStep := 6;
                        ELSIF (nTestStep = 6) AND (nCyclesInPhase >= 140) THEN
                            stHMICommand.eCommandType := CMD_MODE_REQUEST;
                            stHMICommand.eTargetMode := MODE_MANUAL_JOG;
                            stHMICommand.bExecute := TRUE;
                            nTestStep := 7;
                        ELSIF (nTestStep = 7) AND (eCurrentMode = MODE_MANUAL_JOG) THEN
                            eTestPhase := TEST_VERIFY;
                        END_IF

                    9:
                        IF nTestStep = 0 THEN
                            stHMICommand.eCommandType := CMD_MOVE_ABSOLUTE;
                            stHMICommand.nAxisIndex := 1;
                            stHMICommand.fValue1 := 220.0;
                            stHMICommand.fValue2 := 100.0;
                            stHMICommand.bExecute := TRUE;
                            nTestStep := 1;
                        ELSIF (nTestStep = 1) AND (nCyclesInPhase >= 20) THEN
                            GVL_VirtualIO.stVirtualIO.abDriveFault[1] := TRUE;
                            IF (eCurrentMode = MODE_FAULT) AND astAxisStatus[1].bError THEN
                                bFaultObserved := TRUE;
                                GVL_VirtualIO.stVirtualIO.abDriveFault[1] := FALSE;
                                nTestStep := 2;
                            END_IF
                        ELSIF nTestStep = 2 THEN
                            stHMICommand.eCommandType := CMD_RESET;
                            stHMICommand.bExecute := TRUE;
                            nTestStep := 3;
                        ELSIF nTestStep = 3 THEN
                            nTestStep := 4;
                        ELSIF (nTestStep = 4) AND (nCyclesInPhase >= 100) THEN
                            stHMICommand.eCommandType := CMD_RESET_ALL_ALARMS;
                            stHMICommand.bExecute := TRUE;
                            nTestStep := 5;
                        ELSIF nTestStep = 5 THEN
                            nTestStep := 6;
                        ELSIF (nTestStep = 6) AND (nCyclesInPhase >= 150) THEN
                            stHMICommand.eCommandType := CMD_MODE_REQUEST;
                            stHMICommand.eTargetMode := MODE_MANUAL_JOG;
                            stHMICommand.bExecute := TRUE;
                            nTestStep := 7;
                        ELSIF (nTestStep = 7) AND (eCurrentMode = MODE_MANUAL_JOG) THEN
                            eTestPhase := TEST_VERIFY;
                        END_IF

                    10:
                        IF nTestStep = 0 THEN
                            stHMICommand.eCommandType := CMD_MOVE_ABSOLUTE;
                            stHMICommand.nAxisIndex := 1;
                            stHMICommand.fValue1 := 160.0;
                            stHMICommand.fValue2 := 100.0;
                            stHMICommand.bExecute := TRUE;
                            nTestStep := 1;
                        ELSIF (nTestStep = 1) AND (nCyclesInPhase >= 20) THEN
                            GVL_VirtualIO.stVirtualIO.abFollowingError[1] := TRUE;
                            IF (eCurrentMode = MODE_FAULT) AND
                               astAxisStatus[1].bFollowingErrorActive THEN
                                bFaultObserved := TRUE;
                                GVL_VirtualIO.stVirtualIO.abFollowingError[1] := FALSE;
                                nTestStep := 2;
                            END_IF
                        ELSIF nTestStep = 2 THEN
                            stHMICommand.eCommandType := CMD_RESET;
                            stHMICommand.bExecute := TRUE;
                            nTestStep := 3;
                        ELSIF nTestStep = 3 THEN
                            nTestStep := 4;
                        ELSIF (nTestStep = 4) AND (nCyclesInPhase >= 100) THEN
                            stHMICommand.eCommandType := CMD_RESET_ALL_ALARMS;
                            stHMICommand.bExecute := TRUE;
                            nTestStep := 5;
                        ELSIF nTestStep = 5 THEN
                            nTestStep := 6;
                        ELSIF (nTestStep = 6) AND (nCyclesInPhase >= 150) THEN
                            stHMICommand.eCommandType := CMD_MODE_REQUEST;
                            stHMICommand.eTargetMode := MODE_MANUAL_JOG;
                            stHMICommand.bExecute := TRUE;
                            nTestStep := 7;
                        ELSIF (nTestStep = 7) AND (eCurrentMode = MODE_MANUAL_JOG) THEN
                            eTestPhase := TEST_VERIFY;
                        END_IF

                    11:
                        IF nTestStep = 0 THEN
                            stHMICommand.eCommandType := CMD_MOVE_ABSOLUTE;
                            stHMICommand.nAxisIndex := 1;
                            stHMICommand.fValue1 := 140.0;
                            stHMICommand.fValue2 := 100.0;
                            stHMICommand.bExecute := TRUE;
                            nTestStep := 1;
                        ELSIF (nTestStep = 1) AND (nCyclesInPhase >= 20) THEN
                            GVL_VirtualIO.stVirtualIO.abEncoderHealthy[1] := FALSE;
                            IF (eCurrentMode = MODE_FAULT) AND
                               (NOT astAxisStatus[1].bFeedbackHealthy) THEN
                                bFaultObserved := TRUE;
                                GVL_VirtualIO.stVirtualIO.abEncoderHealthy[1] := TRUE;
                                nTestStep := 2;
                            END_IF
                        ELSIF nTestStep = 2 THEN
                            stHMICommand.eCommandType := CMD_RESET;
                            stHMICommand.bExecute := TRUE;
                            nTestStep := 3;
                        ELSIF nTestStep = 3 THEN
                            nTestStep := 4;
                        ELSIF (nTestStep = 4) AND (nCyclesInPhase >= 100) THEN
                            stHMICommand.eCommandType := CMD_RESET_ALL_ALARMS;
                            stHMICommand.bExecute := TRUE;
                            nTestStep := 5;
                        ELSIF nTestStep = 5 THEN
                            nTestStep := 6;
                        ELSIF (nTestStep = 6) AND (nCyclesInPhase >= 150) THEN
                            stHMICommand.eCommandType := CMD_MODE_REQUEST;
                            stHMICommand.eTargetMode := MODE_MANUAL_JOG;
                            stHMICommand.bExecute := TRUE;
                            nTestStep := 7;
                        ELSIF (nTestStep = 7) AND (eCurrentMode = MODE_MANUAL_JOG) THEN
                            eTestPhase := TEST_VERIFY;
                        END_IF

                    12:
                        IF nTestStep = 0 THEN
                            stHMICommand.eCommandType := CMD_MOVE_ABSOLUTE;
                            stHMICommand.nAxisIndex := 1;
                            stHMICommand.fValue1 := 120.0;
                            stHMICommand.fValue2 := 100.0;
                            stHMICommand.bExecute := TRUE;
                            nTestStep := 1;
                        ELSIF (nTestStep = 1) AND (nCyclesInPhase >= 20) THEN
                            GVL_VirtualIO.stVirtualIO.bEtherCATOK := FALSE;
                            IF (eCurrentMode = MODE_FAULT) AND
                               (NOT stSafetyStatus.bNetworkHealthy) THEN
                                bFaultObserved := TRUE;
                                GVL_VirtualIO.stVirtualIO.bEtherCATOK := TRUE;
                                nTestStep := 2;
                            END_IF
                        ELSIF nTestStep = 2 THEN
                            stHMICommand.eCommandType := CMD_RESET;
                            stHMICommand.bExecute := TRUE;
                            nTestStep := 3;
                        ELSIF nTestStep = 3 THEN
                            nTestStep := 4;
                        ELSIF (nTestStep = 4) AND (nCyclesInPhase >= 90) THEN
                            stHMICommand.eCommandType := CMD_RESET_ALL_ALARMS;
                            stHMICommand.bExecute := TRUE;
                            nTestStep := 5;
                        ELSIF nTestStep = 5 THEN
                            nTestStep := 6;
                        ELSIF (nTestStep = 6) AND (nCyclesInPhase >= 140) THEN
                            stHMICommand.eCommandType := CMD_MODE_REQUEST;
                            stHMICommand.eTargetMode := MODE_MANUAL_JOG;
                            stHMICommand.bExecute := TRUE;
                            nTestStep := 7;
                        ELSIF (nTestStep = 7) AND (eCurrentMode = MODE_MANUAL_JOG) THEN
                            eTestPhase := TEST_VERIFY;
                        END_IF

                    13:
                        IF nTestStep = 0 THEN
                            stHMICommand.eCommandType := CMD_STOP;
                            stHMICommand.nAxisIndex := 1;
                            stHMICommand.bExecute := TRUE;
                            nTestStep := 1;
                        ELSIF nCyclesInPhase >= 30 THEN
                            eTestPhase := TEST_VERIFY;
                        END_IF

                    14:
                        GVL_VirtualIO.stVirtualIO.bEStop := TRUE;
                        GVL_VirtualIO.stVirtualIO.bSafetyRelayFB := TRUE;
                        GVL_VirtualIO.stVirtualIO.bGuardDoorClosed := TRUE;
                        GVL_VirtualIO.stVirtualIO.bSTOHealthy := TRUE;
                        GVL_VirtualIO.stVirtualIO.bEtherCATOK := TRUE;
                        GVL_VirtualIO.stVirtualIO.bWatchdogOK := TRUE;
                        GVL_VirtualIO.stVirtualIO.abDriveReady[1] := TRUE;
                        GVL_VirtualIO.stVirtualIO.abDriveFault[1] := FALSE;
                        GVL_VirtualIO.stVirtualIO.abEncoderHealthy[1] := TRUE;
                        IF nCyclesInPhase >= 30 THEN
                            eTestPhase := TEST_VERIFY;
                        END_IF

                    15:
                        IF nTestStep = 0 THEN
                            GVL_VirtualIO.stVirtualIO.bWatchdogOK := FALSE;
                            IF (eCurrentMode = MODE_FAULT) AND
                               (NOT stSafetyStatus.bWatchdogHealthy) THEN
                                bFaultObserved := TRUE;
                                GVL_VirtualIO.stVirtualIO.bWatchdogOK := TRUE;
                                nTestStep := 1;
                            END_IF
                        ELSIF nTestStep = 1 THEN
                            stHMICommand.eCommandType := CMD_RESET;
                            stHMICommand.bExecute := TRUE;
                            nTestStep := 2;
                        ELSIF nTestStep = 2 THEN
                            nTestStep := 3;
                        ELSIF (nTestStep = 3) AND (nCyclesInPhase >= 80) THEN
                            stHMICommand.eCommandType := CMD_RESET_ALL_ALARMS;
                            stHMICommand.bExecute := TRUE;
                            nTestStep := 4;
                        ELSIF nTestStep = 4 THEN
                            nTestStep := 5;
                        ELSIF (nTestStep = 5) AND (nCyclesInPhase >= 130) THEN
                            stHMICommand.eCommandType := CMD_MODE_REQUEST;
                            stHMICommand.eTargetMode := MODE_MANUAL_JOG;
                            stHMICommand.bExecute := TRUE;
                            nTestStep := 6;
                        ELSIF (nTestStep = 6) AND (eCurrentMode = MODE_MANUAL_JOG) THEN
                            eTestPhase := TEST_VERIFY;
                        END_IF

                    16:
                        IF nTestStep = 0 THEN
                            stHMICommand.eCommandType := CMD_MODE_REQUEST;
                            stHMICommand.eTargetMode := MODE_OFF;
                            stHMICommand.bExecute := TRUE;
                            nTestStep := 1;
                        ELSIF nTestStep = 1 THEN
                            nTestStep := 2;
                        ELSIF (nTestStep = 2) AND (nCyclesInPhase >= 30) THEN
                            stHMICommand.eCommandType := CMD_MOVE_ABSOLUTE;
                            stHMICommand.nAxisIndex := 1;
                            stHMICommand.fValue1 := 50.0;
                            stHMICommand.fValue2 := 100.0;
                            stHMICommand.bExecute := TRUE;
                            nTestStep := 3;
                        ELSIF nCyclesInPhase >= 60 THEN
                            eTestPhase := TEST_VERIFY;
                        END_IF
                END_CASE

                IF nCyclesInPhase > 5000 THEN
                    stTestResult.eResult := TRES_TIMEOUT;
                    sActual := 'Test step exceeded 50 second timeout';
                    eTestPhase := TEST_TEARDOWN;
                END_IF

            TEST_VERIFY:
                CASE nCurrentTestID OF
                    1:
                        bVerificationPassed := (eCurrentMode = MODE_MANUAL_JOG) AND
                            astAxisStatus[1].bHomed AND astAxisStatus[2].bHomed;
                        sActual := 'Startup, homing and MANUAL-ready state evaluated';
                    2:
                        bVerificationPassed :=
                            ABS(astAxisStatus[1].fActualPosition - 100.0) <= 0.1;
                        sActual := 'Absolute position tolerance evaluated';
                    3:
                        bVerificationPassed :=
                            ABS(astAxisStatus[1].fActualPosition - fExpectedPosition) <= 0.1;
                        sActual := 'Relative position tolerance evaluated';
                    4:
                        bVerificationPassed := (fPeakPosition > fInitialPosition) AND
                            (fLowPosition < fPeakPosition) AND
                            (NOT astAxisStatus[1].bInMotion);
                        sActual := 'Bidirectional jog displacement and standstill evaluated';
                    5:
                        bVerificationPassed := bFaultObserved AND
                            (eCurrentMode = MODE_MANUAL_JOG) AND stSafetyStatus.bSafeToRun;
                        sActual := 'Positive limit FAULT and recovery evaluated';
                    6:
                        bVerificationPassed := bFaultObserved AND
                            (eCurrentMode = MODE_MANUAL_JOG) AND stSafetyStatus.bSafeToRun;
                        sActual := 'Negative limit FAULT and recovery evaluated';
                    7:
                        bVerificationPassed := bFaultObserved AND
                            (eCurrentMode = MODE_MANUAL_JOG) AND stSafetyStatus.bSafeToRun;
                        sActual := 'E-stop FAULT and recovery evaluated';
                    8:
                        bVerificationPassed := bFaultObserved AND
                            (eCurrentMode = MODE_MANUAL_JOG) AND stSafetyStatus.bSafeToRun;
                        sActual := 'Guard door FAULT and recovery evaluated';
                    9:
                        bVerificationPassed := bFaultObserved AND
                            (eCurrentMode = MODE_MANUAL_JOG) AND
                            (NOT astAxisStatus[1].bError);
                        sActual := 'Drive fault latch and reset evaluated';
                    10:
                        bVerificationPassed := bFaultObserved AND
                            (eCurrentMode = MODE_MANUAL_JOG) AND
                            (NOT astAxisStatus[1].bError);
                        sActual := 'Following error latch and reset evaluated';
                    11:
                        bVerificationPassed := bFaultObserved AND
                            (eCurrentMode = MODE_MANUAL_JOG) AND
                            astAxisStatus[1].bFeedbackHealthy;
                        sActual := 'Encoder feedback loss and reset evaluated';
                    12:
                        bVerificationPassed := bFaultObserved AND
                            (eCurrentMode = MODE_MANUAL_JOG) AND
                            stSafetyStatus.bNetworkHealthy;
                        sActual := 'EtherCAT/network dropout and reset evaluated';
                    13:
                        bVerificationPassed := NOT astAxisStatus[1].bInMotion;
                        sActual := 'Warm restart/stop left axis standstill';
                    14:
                        bVerificationPassed := GVL_VirtualIO.stVirtualIO.bEStop AND
                            GVL_VirtualIO.stVirtualIO.bSafetyRelayFB AND
                            GVL_VirtualIO.stVirtualIO.bGuardDoorClosed AND
                            GVL_VirtualIO.stVirtualIO.bSTOHealthy AND
                            GVL_VirtualIO.stVirtualIO.bEtherCATOK AND
                            GVL_VirtualIO.stVirtualIO.bWatchdogOK AND
                            GVL_VirtualIO.stVirtualIO.abDriveReady[1] AND
                            (NOT GVL_VirtualIO.stVirtualIO.abDriveFault[1]) AND
                            GVL_VirtualIO.stVirtualIO.abEncoderHealthy[1];
                        sActual := 'Virtual cold-start safe defaults evaluated';
                    15:
                        bVerificationPassed := bFaultObserved AND
                            (eCurrentMode = MODE_MANUAL_JOG) AND
                            stSafetyStatus.bWatchdogHealthy;
                        sActual := 'Watchdog timeout FAULT and recovery evaluated';
                    16:
                        bVerificationPassed := (NOT astAxisStatus[1].bInMotion) AND
                            (nActiveAlarmCount > 0);
                        sActual := 'Invalid OFF-state move rejection evaluated';
                END_CASE

                IF bVerificationPassed THEN
                    stTestResult.eResult := TRES_PASS;
                ELSE
                    stTestResult.eResult := TRES_FAIL;
                END_IF
                eTestPhase := TEST_TEARDOWN;

            TEST_TEARDOWN:
                stTestResult.sActual := sActual;
                stTestResult.tDuration := UDINT_TO_TIME(nCyclesInPhase * 10);
                astTestSummary[nCurrentTestID] := stTestResult;
                nTestsRun := nTestsRun + 1;
                IF stTestResult.eResult = TRES_PASS THEN
                    nTestsPassed := nTestsPassed + 1;
                ELSE
                    nTestsFailed := nTestsFailed + 1;
                END_IF

                GVL_VirtualIO.stVirtualIO.bEStop := TRUE;
                GVL_VirtualIO.stVirtualIO.bSafetyRelayFB := TRUE;
                GVL_VirtualIO.stVirtualIO.bGuardDoorClosed := TRUE;
                GVL_VirtualIO.stVirtualIO.bSTOHealthy := TRUE;
                GVL_VirtualIO.stVirtualIO.bEtherCATOK := TRUE;
                GVL_VirtualIO.stVirtualIO.bWatchdogOK := TRUE;
                GVL_VirtualIO.stVirtualIO.abLimitPos[1] := TRUE;
                GVL_VirtualIO.stVirtualIO.abLimitNeg[1] := TRUE;
                GVL_VirtualIO.stVirtualIO.abDriveReady[1] := TRUE;
                GVL_VirtualIO.stVirtualIO.abDriveFault[1] := FALSE;
                GVL_VirtualIO.stVirtualIO.abEncoderHealthy[1] := TRUE;
                GVL_VirtualIO.stVirtualIO.abFollowingError[1] := FALSE;
                stHMICommand.bExecute := FALSE;

                IF bRunSuite AND (nCurrentTestID < 16) THEN
                    nCurrentTestID := nCurrentTestID + 1;
                    eTestPhase := TEST_SETUP;
                    nTestStep := 0;
                    nCyclesInPhase := 0;
                ELSE
                    eTestPhase := TEST_DONE;
                END_IF

            TEST_DONE:
                bTestSuiteRunning := FALSE;
                bTestSuiteComplete := TRUE;
                bRunSuite := FALSE;
                eTestPhase := TEST_IDLE;
        END_CASE
    END_IF
END_IF

END_FUNCTION_BLOCK

(* ---- TraceLogger.st ---- *)
FUNCTION_BLOCK FB_TraceLogger
VAR_INPUT
    bLogEvent : BOOL;
    stEvent : ST_TraceEvent;
    bExportTrigger : BOOL;
    bClearBuffer : BOOL;
END_VAR
VAR_OUTPUT
    nEventCount : UDINT;
    nBufferUsedPercent : UINT;
    bBufferWrapped : BOOL;
    bExportReady : BOOL;
    astRecentEvents : ARRAY[1..20] OF ST_TraceEvent;
END_VAR
VAR
    astRingBuffer : ARRAY[1..1000] OF ST_TraceEvent;
    nWriteIndex : UINT;
    rtrigLog : R_TRIG;
    rtrigExport : R_TRIG;
    rtrigClear : R_TRIG;
    nSourceIndex : DINT;
    nRecentIndex : UINT;
END_VAR

rtrigLog(CLK := bLogEvent);
rtrigExport(CLK := bExportTrigger);
rtrigClear(CLK := bClearBuffer);

IF rtrigClear.Q THEN
    nWriteIndex := 0;
    nEventCount := 0;
    nBufferUsedPercent := 0;
    bBufferWrapped := FALSE;
    bExportReady := FALSE;
    FOR nRecentIndex := 1 TO cTRACE_DISPLAY_COUNT DO
        astRecentEvents[nRecentIndex].nEventID := 0;
        astRecentEvents[nRecentIndex].sDescription := '';
        astRecentEvents[nRecentIndex].fValue := 0.0;
    END_FOR
END_IF

IF rtrigLog.Q THEN
    nWriteIndex := nWriteIndex + 1;
    IF nWriteIndex > cTRACE_BUFFER_SIZE THEN
        nWriteIndex := 1;
        bBufferWrapped := TRUE;
    END_IF
    astRingBuffer[nWriteIndex] := stEvent;
    nEventCount := nEventCount + 1;
END_IF

FOR nRecentIndex := 1 TO cTRACE_DISPLAY_COUNT DO
    nSourceIndex := UINT_TO_DINT(nWriteIndex) - UINT_TO_DINT(nRecentIndex) + 1;
    WHILE nSourceIndex <= 0 DO
        nSourceIndex := nSourceIndex + UINT_TO_DINT(cTRACE_BUFFER_SIZE);
    END_WHILE
    IF (nEventCount >= nRecentIndex) OR bBufferWrapped THEN
        astRecentEvents[nRecentIndex] := astRingBuffer[DINT_TO_UINT(nSourceIndex)];
    END_IF
END_FOR

IF nEventCount >= cTRACE_BUFFER_SIZE THEN
    nBufferUsedPercent := 100;
ELSE
    nBufferUsedPercent := UDINT_TO_UINT(
        (nEventCount * 100) / UINT_TO_UDINT(cTRACE_BUFFER_SIZE)
    );
END_IF

IF rtrigExport.Q THEN
    bExportReady := TRUE;
END_IF

END_FUNCTION_BLOCK

(* ---- AxisManager.st ---- *)
(* ============================================================================
   AxisManager
   Industrial Motion and Safety Bench
   Status: PLACEHOLDER — generated by setup_repo.ps1
   Replace with Claude Code generated content
   ============================================================================ *)

PROGRAM AxisManager
VAR
    (* TODO: Variables will be generated by Claude Code — Prompt 5 *)
END_VAR

(* TODO: Logic will be generated by Claude Code — Prompt 5 *)

END_PROGRAM

(* ---- HomingManager.st ---- *)
(* ============================================================================
   HomingManager
   Industrial Motion and Safety Bench
   Status: PLACEHOLDER — generated by setup_repo.ps1
   Replace with Claude Code generated content
   ============================================================================ *)

PROGRAM HomingManager
VAR
    (* TODO: Variables will be generated by Claude Code — Prompt 5 *)
END_VAR

(* TODO: Logic will be generated by Claude Code — Prompt 5 *)

END_PROGRAM

(* ---- MAIN.st ---- *)
PROGRAM MAIN
VAR
    (* Runtime selection and operator/test controls. *)
    bRunAutomatedTests : BOOL := FALSE;
    bRunSingleTest : BOOL;
    nRequestedTestID : UINT;
    bReloadDefaults : BOOL;
    bTraceExport : BOOL;
    bTraceClear : BOOL;

    (* Portfolio-visible status aliases used by Scope and HMI. *)
    bSimulationRunning : BOOL;
    bSimulationComplete : BOOL;
    bSimulationPassed : BOOL;
    nCurrentTest : UINT;
    nTestsRun : UINT;
    nTestsPassed : UINT;
    nTestsFailed : UINT;
    fActualPosition : LREAL;
    fActualVelocity : LREAL;
    eCurrentMode : E_MachineMode;
    eAxis1State : E_AxisState;
    eLastCommandStatus : E_CommandStatus;
    bSimulationModeActive : BOOL;
    bAxis1InMotion : BOOL;
    bAxis1Error : BOOL;
    nAxis1ErrorCode : UDINT;
    nActiveAlarmCount : UINT;
    nPrimaryAlarmID : UINT;
    nSafetyStatusWord : UINT;

    (* Module instances. *)
    fbConfig : FB_ConfigPackage;
    fbSafety : FB_SafetyManager;
    fbAlarm : FB_AlarmManager;
    fbMode : FB_ModeManager;
    fbCommand : FB_CommandParser;
    fbHoming : FB_HomingManager;
    fbAxis : FB_AxisManager;
    fbTrace : FB_TraceLogger;
    fbHMI : FB_HMIModel;
    fbTest : FB_TestHarness;

    (* NC references are linked to TwinCAT axes for hardware/NC operation.
       They remain unused while bSimulationMode is TRUE. *)
    axis1Ref : AXIS_REF;
    axis2Ref : AXIS_REF;

    (* Inter-module signals. *)
    stSelectedHMICommand : ST_HMICommand;
    abDriveReady : ARRAY[1..2] OF BOOL;
    abHomeSwitchActive : ARRAY[1..2] OF BOOL;
    stTraceEvent : ST_TraceEvent;
    bLogTraceEvent : BOOL;
    ePreviousModeForTrace : E_MachineMode;
    nPreviousAlarmCount : UINT;
    nHeartbeatDivider : UINT;
    bPLCHeartbeat : BOOL;
    nAxis : UINT;
END_VAR

(* 1. Configuration is deterministic and validated before use. *)
fbConfig(bReloadDefaults := bReloadDefaults);

(* 2. Select virtual or physical input image and compute safety permits. *)
IF fbConfig.bSimulationMode THEN
    FOR nAxis := 1 TO cMAX_AXES DO
        abDriveReady[nAxis] := GVL_VirtualIO.stVirtualIO.abDriveReady[nAxis];
    END_FOR
ELSE
    abDriveReady[1] := GVL_IO.bPhysDriveReady1;
    abDriveReady[2] := GVL_IO.bPhysDriveReady2;
END_IF
fbSafety(
    bSimulationMode := fbConfig.bSimulationMode,
    stConfig := fbConfig.stMachineConfig.stSafetyConfig,
    abDriveReady := abDriveReady
);

(* 3. Alarm evaluation intentionally uses the previous scan's axis/homing
      outputs. This gives a deterministic one-scan pipeline without feedback
      loops between AlarmManager and ModeManager. *)
fbAlarm(
    stSafetyStatus := fbSafety.stSafetyStatus,
    bAnyAxisError := fbAxis.bAnyAxisError,
    bHomingError := fbHoming.bHomingError,
    bConfigInvalid := NOT fbConfig.bConfigValid,
    bCommandRejected := fbAxis.bCommandRejected OR
        (fbCommand.eLastCommandStatus = CMDSTAT_ERROR),
    bAckRequested := fbCommand.bAckRequested,
    nAckAlarmID := fbCommand.nAckAlarmID,
    bResetAllRequested := fbCommand.bResetAllRequested
);

(* 4. Machine mode owns state transitions and all operating permits. *)
fbMode(
    stSafetyStatus := fbSafety.stSafetyStatus,
    bAnyFaultActive := fbAlarm.bAnyFaultActive,
    bAllAxesReady := fbAxis.bAllAxesReady,
    bAllAxesHomed := fbHoming.bAllAxesHomed,
    bHomingComplete := fbHoming.bHomingComplete,
    bHomingError := fbHoming.bHomingError,
    eRequestedMode := fbCommand.eRequestedMode,
    bResetRequested := fbCommand.bResetRequested,
    stTimingConfig := fbConfig.stMachineConfig.stTimingConfig
);

(* Automated tests use the same command interface as the HMI. *)
IF fbTest.bTestSuiteRunning THEN
    stSelectedHMICommand := fbTest.stHMICommand;
ELSE
    stSelectedHMICommand := fbHMI.stHMICommand;
END_IF

(* 5. Validate and route the selected command. *)
fbCommand(
    stHMICommand := stSelectedHMICommand,
    eCurrentMode := fbMode.eCurrentMode,
    stModePermits := fbMode.stModePermits,
    stSafetyStatus := fbSafety.stSafetyStatus
);

(* 6. Homing generates abstract seek/set-position requests. *)
IF fbConfig.bSimulationMode THEN
    abHomeSwitchActive := GVL_VirtualIO.stVirtualIO.abHomeSwitch;
ELSE
    abHomeSwitchActive[1] := GVL_IO.bPhysHomeSwitch1;
    abHomeSwitchActive[2] := GVL_IO.bPhysHomeSwitch2;
END_IF

fbHoming(
    eCurrentMode := fbMode.eCurrentMode,
    bStartHoming := fbCommand.bStartHoming,
    bAbortHoming := fbCommand.bAbortHoming,
    abHomeSwitchActive := abHomeSwitchActive,
    astAxisConfig := fbConfig.stMachineConfig.astAxisConfig,
    stTimingConfig := fbConfig.stMachineConfig.stTimingConfig
);

(* 7. AxisManager runs either the deterministic software plant or PLCopen. *)
fbAxis(
    bSimulationMode := fbConfig.bSimulationMode,
    fCycleTimeSeconds := 0.01,
    stModePermits := fbMode.stModePermits,
    eCurrentMode := fbMode.eCurrentMode,
    stCommand := fbCommand.stMotionCommand,
    stSafetyStatus := fbSafety.stSafetyStatus,
    astAxisConfig := fbConfig.stMachineConfig.astAxisConfig,
    abHomeSeekPositive := fbHoming.abSeekPositive,
    abHomeSeekNegative := fbHoming.abSeekNegative,
    abSetHomePosition := fbHoming.abSetPosition,
    afHomePosition := fbHoming.afHomePosition,
    axis1Ref := axis1Ref,
    axis2Ref := axis2Ref
);

(* 8. Generate a compact event stream for important state changes. *)
bLogTraceEvent := FALSE;
IF fbMode.eCurrentMode <> ePreviousModeForTrace THEN
    stTraceEvent.eSource := TRACE_MODE;
    stTraceEvent.nEventID := 100;
    stTraceEvent.sDescription := 'Machine mode changed';
    stTraceEvent.fValue := TO_LREAL(fbMode.eCurrentMode);
    ePreviousModeForTrace := fbMode.eCurrentMode;
    bLogTraceEvent := TRUE;
ELSIF fbAlarm.nActiveAlarmCount <> nPreviousAlarmCount THEN
    stTraceEvent.eSource := TRACE_ALARM;
    stTraceEvent.nEventID := 500;
    stTraceEvent.sDescription := 'Active alarm count changed';
    stTraceEvent.fValue := TO_LREAL(fbAlarm.nActiveAlarmCount);
    nPreviousAlarmCount := fbAlarm.nActiveAlarmCount;
    bLogTraceEvent := TRUE;
ELSIF fbAxis.bMotionComplete THEN
    stTraceEvent.eSource := TRACE_AXIS;
    stTraceEvent.nEventID := 201;
    stTraceEvent.sDescription := 'Axis motion completed';
    stTraceEvent.fValue := fbAxis.astAxisStatus[1].fActualPosition;
    bLogTraceEvent := TRUE;
END_IF

fbTrace(
    bLogEvent := bLogTraceEvent,
    stEvent := stTraceEvent,
    bExportTrigger := bTraceExport,
    bClearBuffer := bTraceClear
);

(* Heartbeat changes every 500 ms for HMI communication supervision. *)
nHeartbeatDivider := nHeartbeatDivider + 1;
IF nHeartbeatDivider >= 50 THEN
    nHeartbeatDivider := 0;
    bPLCHeartbeat := NOT bPLCHeartbeat;
END_IF

(* 9. HMI data is a read-only projection of module outputs. *)
fbHMI(
    eCurrentMode := fbMode.eCurrentMode,
    stModePermits := fbMode.stModePermits,
    astAxisStatus := fbAxis.astAxisStatus,
    stSafetyStatus := fbSafety.stSafetyStatus,
    astActiveAlarms := fbAlarm.astActiveAlarms,
    nActiveAlarmCount := fbAlarm.nActiveAlarmCount,
    eHighestSeverity := fbAlarm.eHighestSeverity,
    astRecentEvents := fbTrace.astRecentEvents,
    eHomingState := fbHoming.eHomingState,
    bSimulationMode := fbConfig.bSimulationMode,
    bPLCHeartbeat := bPLCHeartbeat
);

(* 10. TestHarness is dormant outside simulation mode. *)
fbTest(
    bRunTest := bRunSingleTest,
    nTestID := nRequestedTestID,
    bRunAllTests := bRunAutomatedTests,
    eCurrentMode := fbMode.eCurrentMode,
    astAxisStatus := fbAxis.astAxisStatus,
    stSafetyStatus := fbSafety.stSafetyStatus,
    nActiveAlarmCount := fbAlarm.nActiveAlarmCount,
    nTraceEventCount := fbTrace.nEventCount,
    bSimulationMode := fbConfig.bSimulationMode
);

(* Physical/virtual indication outputs share the same status semantics. *)
IF fbConfig.bSimulationMode THEN
    GVL_VirtualIO.stVirtualIO.bReadyLamp :=
        (fbMode.eCurrentMode = MODE_MANUAL_JOG) OR
        (fbMode.eCurrentMode = MODE_AUTO);
    GVL_VirtualIO.stVirtualIO.bFaultLamp := fbMode.eCurrentMode = MODE_FAULT;
    GVL_VirtualIO.stVirtualIO.bMotionLamp := fbAxis.astAxisStatus[1].bInMotion OR
        fbAxis.astAxisStatus[2].bInMotion;
    GVL_VirtualIO.stVirtualIO.bHomedLamp := fbHoming.bAllAxesHomed;
    GVL_VirtualIO.stVirtualIO.bSafetyRelayCmd := fbSafety.bSafeToRun;
ELSE
    GVL_IO.bPhysReadyLamp :=
        (fbMode.eCurrentMode = MODE_MANUAL_JOG) OR
        (fbMode.eCurrentMode = MODE_AUTO);
    GVL_IO.bPhysFaultLamp := fbMode.eCurrentMode = MODE_FAULT;
    GVL_IO.bPhysMotionLamp := fbAxis.astAxisStatus[1].bInMotion OR
        fbAxis.astAxisStatus[2].bInMotion;
    GVL_IO.bPhysHomedLamp := fbHoming.bAllAxesHomed;
    GVL_IO.bPhysSafetyRelayCmd := fbSafety.bSafeToRun;
END_IF

(* Stable top-level symbols for Scope, ADS clients, and portfolio demos. *)
bSimulationRunning := fbTest.bTestSuiteRunning;
bSimulationComplete := fbTest.bTestSuiteComplete;
bSimulationPassed := fbTest.bTestSuiteComplete AND (fbTest.nTestsFailed = 0);
nCurrentTest := fbTest.nCurrentTestID;
nTestsRun := fbTest.nTestsRun;
nTestsPassed := fbTest.nTestsPassed;
nTestsFailed := fbTest.nTestsFailed;
fActualPosition := fbAxis.astAxisStatus[1].fActualPosition;
fActualVelocity := fbAxis.astAxisStatus[1].fActualVelocity;
eCurrentMode := fbMode.eCurrentMode;
eAxis1State := fbAxis.astAxisStatus[1].eAxisState;
eLastCommandStatus := fbCommand.eLastCommandStatus;
bSimulationModeActive := fbConfig.bSimulationMode;
bAxis1InMotion := fbAxis.astAxisStatus[1].bInMotion;
bAxis1Error := fbAxis.astAxisStatus[1].bError;
nAxis1ErrorCode := fbAxis.astAxisStatus[1].nErrorCode;
nActiveAlarmCount := fbAlarm.nActiveAlarmCount;
nPrimaryAlarmID := 0;
IF fbAlarm.nActiveAlarmCount > 0 THEN
    nPrimaryAlarmID := fbAlarm.astActiveAlarms[1].nID;
END_IF
nSafetyStatusWord := fbSafety.stSafetyStatus.nSafetyStatusWord;

END_PROGRAM
